Staubli VAL3: Control_PanelB.pgx

public program Control_PanelB(string x_sLeftTitle, string x_sRightTitle)
begin

  //画左右两个方框

  call Control_PanelS(x_sLeftTitle,0,0,18,11)

  call Control_PanelS(x_sRightTitle,20,0,18,11)

end
